// TIA Portal V20 export
// export: Created 2025-12-01T14:57:44.4127247Z, ExportSetting None, DisplayName Totally Integrated Automation Portal, DisplayVersion V20 Update 3, DisplayName TIA Portal Openness, DisplayVersion V20 Update 3, DisplayName TIA Portal Version Control Interface, DisplayVersion V20 Update 3, DisplayName STEP 7 Professional, DisplayVersion V20 Update 3, DisplayName STEP 7 Safety, DisplayVersion V20 Update 2, DisplayName WinCC Basic/Comfort/Advanced, DisplayVersion V20 Update 3, DisplayName WinCC Professional, DisplayVersion V20 Update 3, DisplayName WinCC Unified, DisplayVersion V20 Update 3
FUNCTION "FC534_Estados_ocupacion_V2" : Void   // FC534, LAD
{ S7_Optimized_Access := 'TRUE' }
// stored: AutoNumber false, SetENOAutomatically false
   VAR_INPUT
      NumeroMesa : UInt;   // Numero de Mesa
      Phs_1 : Bool;
      Phs_2 : Bool;
      Phs_3 : Bool;
      Phs_4 : Bool;
      Tiempo_Ocupado : UDInt;
      ATRIBUTO_NIVEL_1 : String;   // 0
      ATRIBUTO_NIVEL_2 : String;   // 25
      ATRIBUTO_NIVEL_3 : String;   // 50
      ATRIBUTO_NIVEL_4 : String;   // 75
      ATRIBUTO_NIVEL_5 : String;   // 100
   END_VAR
   VAR_IN_OUT
      DB_Eventos : Array[*] of Char;
      MemEstadoOcupa : Byte;   // Memoria del ultimo estado emitido
      Memorias_ocupacion : Int;
   END_VAR
   VAR_TEMP
      Emitir : Bool;
      Nuevo_estado : Byte;
      VarEvento : Struct
         InicioEventos : UInt;
         FinalEventos : UInt;
         Indice : UInt;
         Posicion_Inicial : UInt;
         CNT_Chars : UInt;
         Motivo : UInt;
         Mesa_String : String;
         Evento : String;
         Encontrado : Bool;
         Motivo_string : String;
      END_STRUCT;
   END_VAR
BEGIN

REGION Network 1: si el sistema no está en marcha o hacemos un reset, borramos la memoria del estado para que se vuelva a emitir
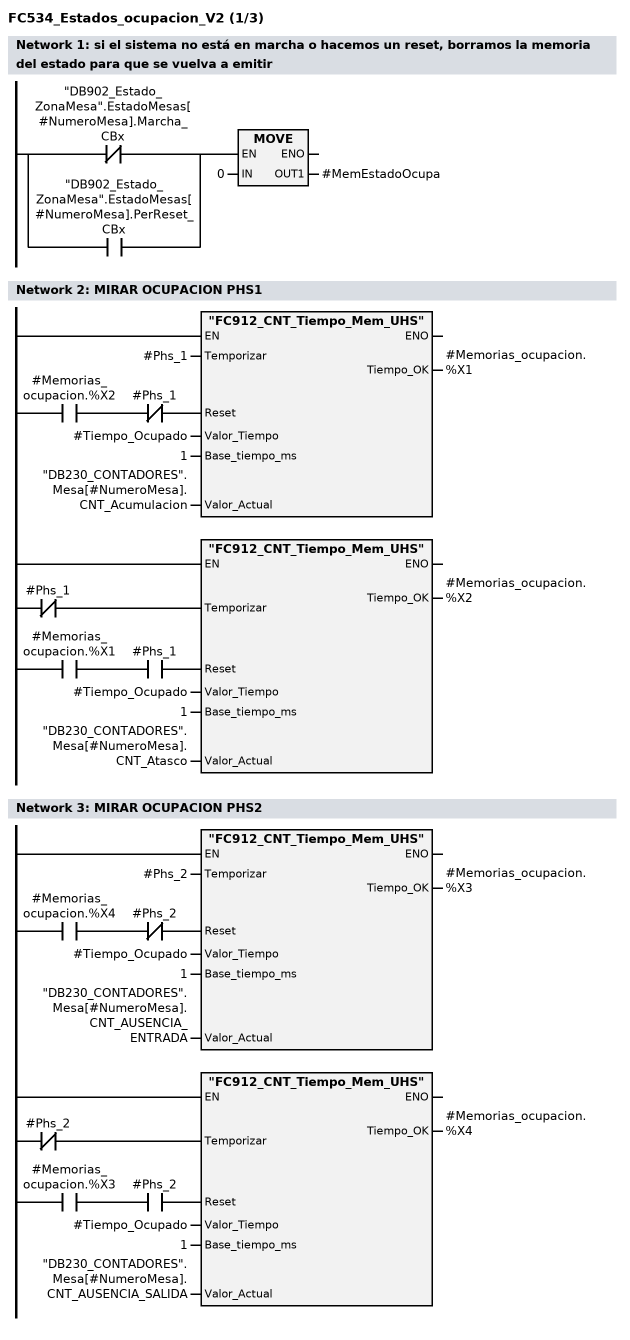
   RUNG wire#powerrail
      I_Contact( "DB902_Estado_ZonaMesa".EstadoMesas[#NumeroMesa].Marcha_CBx )
      wire#w1
      Move(in := 0, out1 => #MemEstadoOcupa)
   END_RUNG
   RUNG wire#powerrail
      Contact( "DB902_Estado_ZonaMesa".EstadoMesas[#NumeroMesa].PerReset_CBx )
   END_RUNG wire#w1
   // the same network as SCL:
   IF NOT "DB902_Estado_ZonaMesa".EstadoMesas[#NumeroMesa].Marcha_CBx OR "DB902_Estado_ZonaMesa".EstadoMesas[#NumeroMesa].PerReset_CBx THEN
       #MemEstadoOcupa := 0;
   END_IF;
END_REGION

REGION Network 2: MIRAR OCUPACION PHS1
   RUNG wire#powerrail
      "FC912_CNT_Tiempo_Mem_UHS"(Reset := wire#w1, Temporizar := #Phs_1, Valor_Tiempo := #Tiempo_Ocupado, Base_tiempo_ms := 1, Valor_Actual := "DB230_CONTADORES".Mesa[#NumeroMesa].CNT_Acumulacion, Tiempo_OK => #Memorias_ocupacion.%X1)
   END_RUNG
   RUNG wire#powerrail
      Contact( #Memorias_ocupacion.%X2 )
      I_Contact( #Phs_1 )
   END_RUNG wire#w1
   RUNG wire#powerrail
      "FC912_CNT_Tiempo_Mem_UHS"(Temporizar := wire#w2, Reset := wire#w3, Valor_Tiempo := #Tiempo_Ocupado, Base_tiempo_ms := 1, Valor_Actual := "DB230_CONTADORES".Mesa[#NumeroMesa].CNT_Atasco, Tiempo_OK => #Memorias_ocupacion.%X2)
   END_RUNG
   RUNG wire#powerrail
      I_Contact( #Phs_1 )
   END_RUNG wire#w2
   RUNG wire#powerrail
      Contact( #Memorias_ocupacion.%X1 )
      Contact( #Phs_1 )
   END_RUNG wire#w3
   // the same network as SCL:
   "FC912_CNT_Tiempo_Mem_UHS"(Temporizar := #Phs_1,
                           Reset := #Memorias_ocupacion.%X2 AND NOT #Phs_1,
                           Valor_Tiempo := #Tiempo_Ocupado,
                           Base_tiempo_ms := 1,
                           Valor_Actual := "DB230_CONTADORES".Mesa[#NumeroMesa].CNT_Acumulacion,
                           Tiempo_OK => #Memorias_ocupacion.%X1);
   "FC912_CNT_Tiempo_Mem_UHS"(Temporizar := NOT #Phs_1,
                           Reset := #Memorias_ocupacion.%X1 AND #Phs_1,
                           Valor_Tiempo := #Tiempo_Ocupado,
                           Base_tiempo_ms := 1,
                           Valor_Actual := "DB230_CONTADORES".Mesa[#NumeroMesa].CNT_Atasco,
                           Tiempo_OK => #Memorias_ocupacion.%X2);
END_REGION

REGION Network 3: MIRAR OCUPACION PHS2
   RUNG wire#powerrail
      "FC912_CNT_Tiempo_Mem_UHS"(Reset := wire#w1, Temporizar := #Phs_2, Valor_Tiempo := #Tiempo_Ocupado, Base_tiempo_ms := 1, Valor_Actual := "DB230_CONTADORES".Mesa[#NumeroMesa].CNT_AUSENCIA_ENTRADA, Tiempo_OK => #Memorias_ocupacion.%X3)
   END_RUNG
   RUNG wire#powerrail
      Contact( #Memorias_ocupacion.%X4 )
      I_Contact( #Phs_2 )
   END_RUNG wire#w1
   RUNG wire#powerrail
      "FC912_CNT_Tiempo_Mem_UHS"(Temporizar := wire#w2, Reset := wire#w3, Valor_Tiempo := #Tiempo_Ocupado, Base_tiempo_ms := 1, Valor_Actual := "DB230_CONTADORES".Mesa[#NumeroMesa].CNT_AUSENCIA_SALIDA, Tiempo_OK => #Memorias_ocupacion.%X4)
   END_RUNG
   RUNG wire#powerrail
      I_Contact( #Phs_2 )
   END_RUNG wire#w2
   RUNG wire#powerrail
      Contact( #Memorias_ocupacion.%X3 )
      Contact( #Phs_2 )
   END_RUNG wire#w3
   // the same network as SCL:
   "FC912_CNT_Tiempo_Mem_UHS"(Temporizar := #Phs_2,
                           Reset := #Memorias_ocupacion.%X4 AND NOT #Phs_2,
                           Valor_Tiempo := #Tiempo_Ocupado,
                           Base_tiempo_ms := 1,
                           Valor_Actual := "DB230_CONTADORES".Mesa[#NumeroMesa].CNT_AUSENCIA_ENTRADA,
                           Tiempo_OK => #Memorias_ocupacion.%X3);
   "FC912_CNT_Tiempo_Mem_UHS"(Temporizar := NOT #Phs_2,
                           Reset := #Memorias_ocupacion.%X3 AND #Phs_2,
                           Valor_Tiempo := #Tiempo_Ocupado,
                           Base_tiempo_ms := 1,
                           Valor_Actual := "DB230_CONTADORES".Mesa[#NumeroMesa].CNT_AUSENCIA_SALIDA,
                           Tiempo_OK => #Memorias_ocupacion.%X4);
END_REGION

REGION Network 4: MIRAR OCUPACION PHS3
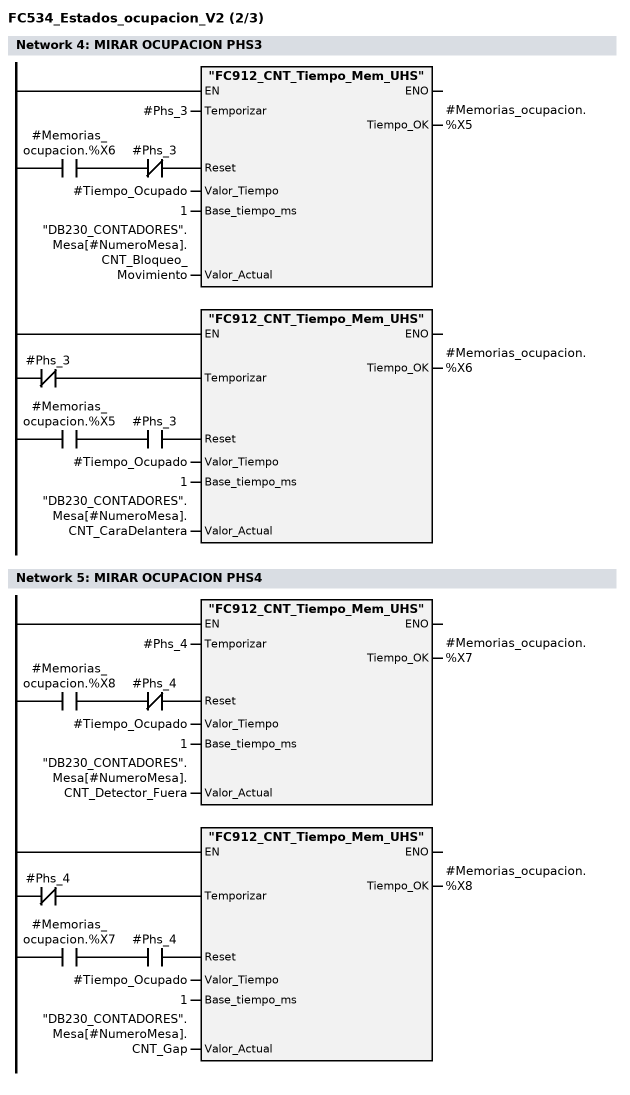
   RUNG wire#powerrail
      "FC912_CNT_Tiempo_Mem_UHS"(Reset := wire#w1, Temporizar := #Phs_3, Valor_Tiempo := #Tiempo_Ocupado, Base_tiempo_ms := 1, Valor_Actual := "DB230_CONTADORES".Mesa[#NumeroMesa].CNT_Bloqueo_Movimiento, Tiempo_OK => #Memorias_ocupacion.%X5)
   END_RUNG
   RUNG wire#powerrail
      Contact( #Memorias_ocupacion.%X6 )
      I_Contact( #Phs_3 )
   END_RUNG wire#w1
   RUNG wire#powerrail
      "FC912_CNT_Tiempo_Mem_UHS"(Temporizar := wire#w2, Reset := wire#w3, Valor_Tiempo := #Tiempo_Ocupado, Base_tiempo_ms := 1, Valor_Actual := "DB230_CONTADORES".Mesa[#NumeroMesa].CNT_CaraDelantera, Tiempo_OK => #Memorias_ocupacion.%X6)
   END_RUNG
   RUNG wire#powerrail
      I_Contact( #Phs_3 )
   END_RUNG wire#w2
   RUNG wire#powerrail
      Contact( #Memorias_ocupacion.%X5 )
      Contact( #Phs_3 )
   END_RUNG wire#w3
   // the same network as SCL:
   "FC912_CNT_Tiempo_Mem_UHS"(Temporizar := #Phs_3,
                           Reset := #Memorias_ocupacion.%X6 AND NOT #Phs_3,
                           Valor_Tiempo := #Tiempo_Ocupado,
                           Base_tiempo_ms := 1,
                           Valor_Actual := "DB230_CONTADORES".Mesa[#NumeroMesa].CNT_Bloqueo_Movimiento,
                           Tiempo_OK => #Memorias_ocupacion.%X5);
   "FC912_CNT_Tiempo_Mem_UHS"(Temporizar := NOT #Phs_3,
                           Reset := #Memorias_ocupacion.%X5 AND #Phs_3,
                           Valor_Tiempo := #Tiempo_Ocupado,
                           Base_tiempo_ms := 1,
                           Valor_Actual := "DB230_CONTADORES".Mesa[#NumeroMesa].CNT_CaraDelantera,
                           Tiempo_OK => #Memorias_ocupacion.%X6);
END_REGION

REGION Network 5: MIRAR OCUPACION PHS4
   RUNG wire#powerrail
      "FC912_CNT_Tiempo_Mem_UHS"(Reset := wire#w1, Temporizar := #Phs_4, Valor_Tiempo := #Tiempo_Ocupado, Base_tiempo_ms := 1, Valor_Actual := "DB230_CONTADORES".Mesa[#NumeroMesa].CNT_Detector_Fuera, Tiempo_OK => #Memorias_ocupacion.%X7)
   END_RUNG
   RUNG wire#powerrail
      Contact( #Memorias_ocupacion.%X8 )
      I_Contact( #Phs_4 )
   END_RUNG wire#w1
   RUNG wire#powerrail
      "FC912_CNT_Tiempo_Mem_UHS"(Temporizar := wire#w2, Reset := wire#w3, Valor_Tiempo := #Tiempo_Ocupado, Base_tiempo_ms := 1, Valor_Actual := "DB230_CONTADORES".Mesa[#NumeroMesa].CNT_Gap, Tiempo_OK => #Memorias_ocupacion.%X8)
   END_RUNG
   RUNG wire#powerrail
      I_Contact( #Phs_4 )
   END_RUNG wire#w2
   RUNG wire#powerrail
      Contact( #Memorias_ocupacion.%X7 )
      Contact( #Phs_4 )
   END_RUNG wire#w3
   // the same network as SCL:
   "FC912_CNT_Tiempo_Mem_UHS"(Temporizar := #Phs_4,
                           Reset := #Memorias_ocupacion.%X8 AND NOT #Phs_4,
                           Valor_Tiempo := #Tiempo_Ocupado,
                           Base_tiempo_ms := 1,
                           Valor_Actual := "DB230_CONTADORES".Mesa[#NumeroMesa].CNT_Detector_Fuera,
                           Tiempo_OK => #Memorias_ocupacion.%X7);
   "FC912_CNT_Tiempo_Mem_UHS"(Temporizar := NOT #Phs_4,
                           Reset := #Memorias_ocupacion.%X7 AND #Phs_4,
                           Valor_Tiempo := #Tiempo_Ocupado,
                           Base_tiempo_ms := 1,
                           Valor_Actual := "DB230_CONTADORES".Mesa[#NumeroMesa].CNT_Gap,
                           Tiempo_OK => #Memorias_ocupacion.%X8);
END_REGION

REGION Network 6: generar el nuevo estado a emitir
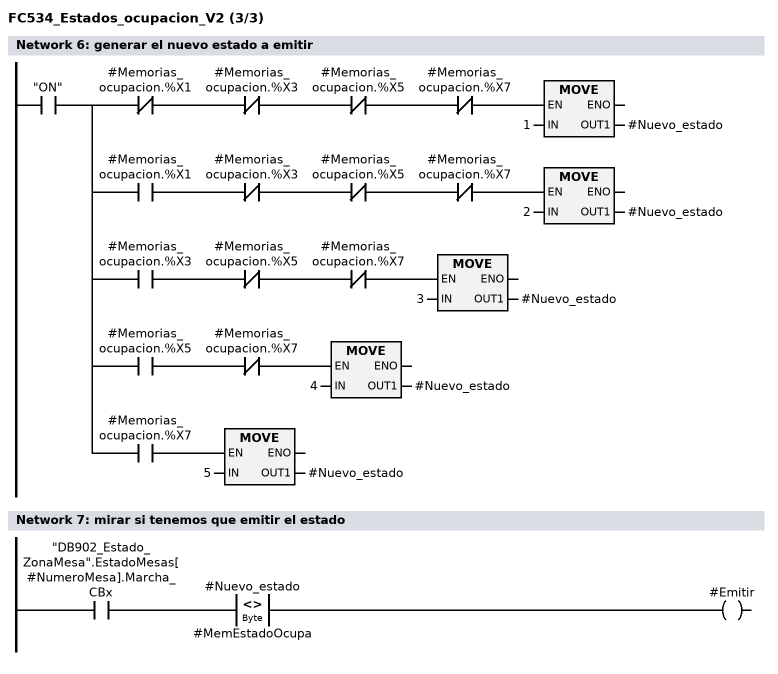
   RUNG wire#powerrail
      Contact( "ON" )
      wire#w1
      I_Contact( #Memorias_ocupacion.%X1 )
      I_Contact( #Memorias_ocupacion.%X3 )
      I_Contact( #Memorias_ocupacion.%X5 )
      I_Contact( #Memorias_ocupacion.%X7 )
      Move(in := 1, out1 => #Nuevo_estado)
   END_RUNG
   RUNG wire#w1
      Contact( #Memorias_ocupacion.%X1 )
      I_Contact( #Memorias_ocupacion.%X3 )
      I_Contact( #Memorias_ocupacion.%X5 )
      I_Contact( #Memorias_ocupacion.%X7 )
      Move(in := 2, out1 => #Nuevo_estado)
   END_RUNG
   RUNG wire#w1
      Contact( #Memorias_ocupacion.%X3 )
      I_Contact( #Memorias_ocupacion.%X5 )
      I_Contact( #Memorias_ocupacion.%X7 )
      Move(in := 3, out1 => #Nuevo_estado)
   END_RUNG
   RUNG wire#w1
      Contact( #Memorias_ocupacion.%X5 )
      I_Contact( #Memorias_ocupacion.%X7 )
      Move(in := 4, out1 => #Nuevo_estado)
   END_RUNG
   RUNG wire#w1
      Contact( #Memorias_ocupacion.%X7 )
      Move(in := 5, out1 => #Nuevo_estado)
   END_RUNG
   // the same network as SCL:
   IF "ON" AND NOT #Memorias_ocupacion.%X1 AND NOT #Memorias_ocupacion.%X3 AND NOT #Memorias_ocupacion.%X5 AND NOT #Memorias_ocupacion.%X7 THEN
       #Nuevo_estado := 1;
   END_IF;
   IF "ON" AND #Memorias_ocupacion.%X1 AND NOT #Memorias_ocupacion.%X3 AND NOT #Memorias_ocupacion.%X5 AND NOT #Memorias_ocupacion.%X7 THEN
       #Nuevo_estado := 2;
   END_IF;
   IF "ON" AND #Memorias_ocupacion.%X3 AND NOT #Memorias_ocupacion.%X5 AND NOT #Memorias_ocupacion.%X7 THEN
       #Nuevo_estado := 3;
   END_IF;
   IF "ON" AND #Memorias_ocupacion.%X5 AND NOT #Memorias_ocupacion.%X7 THEN #Nuevo_estado := 4; END_IF;
   IF "ON" AND #Memorias_ocupacion.%X7 THEN #Nuevo_estado := 5; END_IF;
END_REGION

REGION Network 7: mirar si tenemos que emitir el estado
   RUNG wire#powerrail
      Contact( "DB902_Estado_ZonaMesa".EstadoMesas[#NumeroMesa].Marcha_CBx )
      { S7_Templates := "SrcType := Byte" } NE_Contact(in1 := #Nuevo_estado, in2 := #MemEstadoOcupa)
      Coil( #Emitir )
   END_RUNG
   // the same network as SCL:
   #Emitir := "DB902_Estado_ZonaMesa".EstadoMesas[#NumeroMesa].Marcha_CBx AND (#Nuevo_estado <> #MemEstadoOcupa);
END_REGION

REGION Network 8 (SCL): EMISION DEL EVENTO PRES CON LOS ATRIBUTOS DEL GALIBO DEFINIDOS

   REGION EnvioEvento_PRES
       //////////////////////////////////////////////////////////////////////////////
       // Envio de Evento
       IF #Emitir = TRUE THEN
           //Inicializacion de Variables de Emision. Busca el limite inferior y superior del array
           #VarEvento.InicioEventos := DINT_TO_UINT(LOWER_BOUND(ARR := #DB_Eventos, DIM := 1));
           #VarEvento.FinalEventos := DINT_TO_UINT(UPPER_BOUND(ARR := #DB_Eventos, DIM := 1));

           #VarEvento.Encontrado := FALSE;
           #VarEvento.Posicion_Inicial := 0;
           #VarEvento.Evento := DELETE(IN := #VarEvento.Evento, L := 255, P := 1);

           // Conversion de numero de mesa
           #VarEvento.Mesa_String := UINT_TO_STRING(#NumeroMesa + "CTE_OffsetMesa");
           #VarEvento.Mesa_String := DELETE(IN := #VarEvento.Mesa_String, L := 1, P := 1); //Se elimnia el caracter '+' que genera la conversion


           // Busqueda del ultimo caracter de emision "0x00" en el DB de emision
           FOR #VarEvento.Indice := #VarEvento.InicioEventos TO #VarEvento.FinalEventos DO
               IF #DB_Eventos[#VarEvento.Indice] = BYTE#0 THEN
                   #VarEvento.Posicion_Inicial := #VarEvento.Indice;
                   #VarEvento.Encontrado := TRUE;
                   EXIT;
               END_IF;
           END_FOR;


           //NIEVES, MIRAR AQUI COMO FORMATEAR LA COMA SI NO ES EL PRIMER EVENTO
           //

           #VarEvento.Motivo := #Nuevo_estado;


               CASE  #VarEvento.Motivo OF
                   1:  // motivo normal
                       #VarEvento.Motivo_string := #ATRIBUTO_NIVEL_1;
                   2:  // motivo reset
                       #VarEvento.Motivo_string := #ATRIBUTO_NIVEL_2;
                       ;
                   3:  // motivo normal
                       #VarEvento.Motivo_string := #ATRIBUTO_NIVEL_3;
                   4:  // motivo reset
                       #VarEvento.Motivo_string := #ATRIBUTO_NIVEL_4;
                   5:  // motivo reset
                       #VarEvento.Motivo_string := #ATRIBUTO_NIVEL_5;
                       ;
                   ELSE  // Statement section ELSE
                       #VarEvento.Motivo_string := '';
               END_CASE;

   //------------------------------------------------------------------------------------------------

           // Enviar el Evento
               IF #VarEvento.Encontrado = TRUE AND #VarEvento.Posicion_Inicial <= "JDT1_MaxBytes" THEN

                   IF #VarEvento.Indice <> 0 THEN
                       #DB_Eventos[#VarEvento.Posicion_Inicial] := ',';
                       #VarEvento.Posicion_Inicial := #VarEvento.Posicion_Inicial + 1;
                   END_IF;

               //Creacion de la cadena a enviar
               #VarEvento.Evento := CONCAT(IN1 := '{DIDA',
                                           IN2 := '[TIPO]MESA[NUME]', IN3 :=  #VarEvento.Mesa_String,
                                           IN4 := '[FULL]', IN5 :=  #VarEvento.Motivo_string,
                                           IN6 := '}');

               //Conversion a char y envio
               Strg_TO_Chars(Strg := #VarEvento.Evento,
                             pChars := #VarEvento.Posicion_Inicial,
                             Cnt => #VarEvento.CNT_Chars,
                             Chars := #DB_Eventos);
               #MemEstadoOcupa := #Nuevo_estado;


           END_IF;
       END_IF;

   END_REGION
END_REGION
END_FUNCTION
